Staubli VAL3: refreshStatic.pgx

program refreshStatic()
  local string l_sMessage
  local num i
begin
  cls()
  //
  // set the view of the page..
  //
  // SET THE PAGE NUMBER
  use:nPage=1010
  // USE <>PROFILE for <>PAGE
  use:nPage=use:nPage+abs(limit(saveData:mode,0,2)-2)
  if cycleStatus:bCycle
    use:nPage=use:nPage+3
  endIf
  // load the menu page
  if saveData:language!="japanese"
    // SET THE VIEW OF THE PAGE
    call language:page(l_sMessage,use:nPage)
    // define the menu
    call use:stringToArray(l_sMessage,sMenu)
  else
    // japanese use the array for the menu
    call language:page(sMenu8,use:nPage)
    call use:stringCopy(sMenu8,sMenu)
  endIf
  //
  // polymorphism
  //
  // get the user Menu or special one
  call trajType:getFunctionSel(sMenuUser)
  // OVERRIDE
  for i=0 to size(sMenuUser)-1
    if sMenuUser[i]!=""
      sMenu[i]=sMenuUser[i]
    endIf
  endFor
  // set the menu
  if saveData:language!="japanese"
    call use:setMenu(sMenu,true,3)
  else
    call use:setMenu(sMenu,false,3)
  endIf
  call use:getMenu(sMenu,bButton)
  //
  // CREATE THE LIST
  //
  // define your list size for default
  call use:setSizeList(19,0,19,11)
  call use:setView(bLarge)
  //
  call use:listcreate(saveData:sTrajTypeUsing)
  //
  call use:listadd(sList)
  //
  // refresh the list
  call use:selectNewField(nSelected,nIndex,nView)
  //
  // is a filter using ??
  if  saveData:sTrajFilter!=""
    call language:message(l_sMessage,64)
    call use:type(0,1,l_sMessage+">"+saveData:sTrajFilter)
  else
    // clean
    call use:typeLen(0,1," ",use:nBottomX)
  endIf
end
